FUNCTION_BLOCK FBUO_OverPressure
VAR_INPUT
    fbOPprocessState 		: BOOL;
    fbValvePositionReady 	: BOOL;
	fbPumpActive 			: BOOL;
	fbPumpSpeed				: REAL;
END_VAR
VAR_IN_OUT
    fbValves : ARRAY[1..GVL.valveCount] OF ST_Valves;
END_VAR
VAR_OUTPUT
	
END_VAR
VAR
    valveIndexOpen : ARRAY[1..GVL.valveCount] OF INT := [2,5];
	numValvesToOpen : INT := 10;
	valveIndexClose : ARRAY[1..GVL.valveCount] OF INT := [2,5];
	numValvesToClose : INT := 10;
    targetState : INT;
    targetOpenClose : BOOL;
	fbValvePos : FB_ValvePOS;
	valveCtrl : FB_valveCTRL;
	valveIndex: INT;
END_VAR

IF fbOPprocessState THEN
	
	fbValvePos(fbValveIndexOpen := valveIndexOpen,
            fbNumValvesToOpen := numValvesToOpen,
			fbValveIndexClose := valveIndexClose,
            fbNumValvesToClose := numValvesToClose,
            fbValves := fbValves,
			fbProcessValves2Open := fbValvePositionReady);
    
    ValveCtrl(fbValves := fbValves);
    IO.AO1_dilutionSV := fbValves[1].AO1;
    IO.AO1_wfiSV := fbValves[2].AO1;
    IO.AO1_formDrain := fbValves[3].AO1;
    IO.AO1_wfiBypassIn := fbValves[4].AO1;
	IO.AO1_wfiFilterIn := fbValves[5].AO1;
	IO.AO1_wfiFilterOut := fbValves[6].AO1;
	IO.AO1_wfiBypassOut := fbValves[7].AO1;
	IO.AO1_dilutionDiV := fbValves[8].AO1;
	IO.AO1_FormManifold := fbValves[9].AO1;
	IO.AO1_SuspManifold := fbValves[10].AO1;
	
	
	
//-----------------------PUMP Control ----------------------//	
// 	IF fbPumpActive THEN
// 	outputAO3 := IO.AO3 := 5;
// 		GVL.DO_wfiPump := fbPumpActive;
// 		GVL.AO_wfiPump := fbPumpSpeed;
// 	ELSE
// 		GVL.DO_wfiPump := fbPumpActive;
// 		GVL.AO_wfiPump := 0;
// 	END_IF	
//---------------------------------------------------------//	
END_IF

END_FUNCTION_BLOCK

(* stored: Version 1.1.0.1
   POU FBUO_OverPressure: Id {d0d6383a-d8b4-0693-144b-0eb7d3fc8ac4}, SpecialFunc None *)
